{attribute 'qualified_only'}
VAR_GLOBAL



END_VAR

(* stored: Version 1.1.0.1, ProductVersion 3.1.4022.12
   GVL GVL: Id {be9d8fe6-ccef-49b4-a0d9-87455acac8e5} *)
